FUNCTION_BLOCK FB_MovingAverage
VAR
    _StorageArray : POINTER TO LREAL;
    _FilterSize : UINT;

    Index : INT := -1;
    Average, Sum : LREAL;

    EqualOrMoreDataPointsThanFilterSize : BOOL := FALSE;
END_VAR

METHOD PUBLIC AddDataPoint
VAR_INPUT
    x : LREAL;
END_VAR
Index := (Index + 1) MOD UINT_TO_INT(_FilterSize);

Sum := Sum - _StorageArray[Index];
_StorageArray[Index] := x;
Sum := Sum + x;

IF NOT EqualOrMoreDataPointsThanFilterSize AND (Index = (UINT_TO_INT(_FilterSize) - 1)) THEN
    EqualOrMoreDataPointsThanFilterSize := TRUE;
END_IF

IF EqualOrMoreDataPointsThanFilterSize THEN
    Average := Sum / UINT_TO_LREAL(_FilterSize);
ELSE
    Average := Sum / INT_TO_LREAL(Index + 1);
END_IF
END_METHOD

METHOD FB_init : BOOL
VAR_INPUT
	bInitRetains : BOOL; // if TRUE, the retain variables are initialized (warm start / cold start)
	bInCopyCode : BOOL;  // if TRUE, the instance afterwards gets moved into the copy code (online change)
    StorageArray : POINTER TO LREAL;
    FilterSize : UINT;
END_VAR
_StorageArray := StorageArray;
_FilterSize := FilterSize;
END_METHOD

METHOD PUBLIC GetAverage : LREAL
GetAverage := Average;
END_METHOD

END_FUNCTION_BLOCK

(* stored: Version 1.1.0.1, ProductVersion 3.1.4022.16
   POU FB_MovingAverage: Id {b42e9e0a-d273-4f14-b645-26e0c449a8fe}, SpecialFunc None
   Method AddDataPoint: Id {6ea6bd01-6552-44a7-b6e5-6523e96a3028}
   Method FB_init: Id {488b24e6-9756-4bc4-9cad-9b96bc26d0ca}
   Method GetAverage: Id {8cc88594-ce31-4168-81ef-34c900512645} *)
